// TwinCAT 3 PLC project Tests
// ProgramVersion: 3.1.4023.0
// libraries:
//   Tc2_Standard, * (Beckhoff Automation GmbH)
//   Tc2_System, * (Beckhoff Automation GmbH)
//   Tc3_Module, * (Beckhoff Automation GmbH)
// project tree:
//   DUTs/Alias/ T_Bool.TcDUT, T_Enum.TcDUT, T_SimpleStruct.TcDUT, T_PackedFb.TcDUT, T_String.TcDUT, T_Lreal.TcDUT, T_Dint.TcDUT, T_Wstring.TcDUT
//   DUTs/Enums/ E_Enum.TcDUT
//   DUTs/Struct/ ST_Simple.TcDUT, ST_Packed.TcDUT, ST_Complex.TcDUT, ST_STRUCT.TcDUT
//   DUTs/Unions/ U_Simple.TcDUT
//   / PlcTask.TcTTO
//   POUs/FBs/ FB_Invokable.TcPOU, FB_Simple.TcPOU, FB_Complex.TcPOU, FB_Packed.TcPOU
//   POUs/ P_Benchmark.TcPOU, P_Invoke.TcPOU, P_Notifications.TcPOU, P_Read.TcPOU, P_Write.TcPOU
// real-time tasks:
//   TASK PlcTask: cycle T#10ms, priority 8, ADS port 350
//   TASK FreeTask: cycle T#10ms, priority 6, ADS port 301

CONFIGURATION Tests
    RESOURCE PLC ON TwinCAT3
        TASK PlcTask(INTERVAL := T#10ms, PRIORITY := 8);
        PROGRAM P_Read WITH PlcTask : P_Read;
        PROGRAM P_Write WITH PlcTask : P_Write;
        PROGRAM P_Invoke WITH PlcTask : P_Invoke;
        PROGRAM P_Notifications WITH PlcTask : P_Notifications;
        PROGRAM P_Benchmark WITH PlcTask : P_Benchmark;
    END_RESOURCE
END_CONFIGURATION

// ---- DUTs/Alias/T_Bool.TcDUT
TYPE T_Bool : BOOL; END_TYPE

// ---- DUTs/Alias/T_Enum.TcDUT
TYPE T_Enum : E_Enum; END_TYPE

// ---- DUTs/Alias/T_SimpleStruct.TcDUT
TYPE T_SimpleStruct : ST_Simple; END_TYPE

// ---- DUTs/Alias/T_PackedFb.TcDUT
TYPE T_PackedFb : FB_Packed; END_TYPE

// ---- DUTs/Alias/T_String.TcDUT
TYPE T_String : STRING; END_TYPE

// ---- DUTs/Alias/T_Lreal.TcDUT
TYPE T_Lreal : LREAL; END_TYPE

// ---- DUTs/Alias/T_Dint.TcDUT
TYPE T_Dint : DINT; END_TYPE

// ---- DUTs/Alias/T_Wstring.TcDUT
TYPE T_Wstring : WSTRING; END_TYPE

// ---- DUTs/Enums/E_Enum.TcDUT
{attribute 'qualified_only'}
{attribute 'strict'}
TYPE E_Enum :
(
	Member0 := 0,
	Member1,
	Member2
);
END_TYPE

// ---- DUTs/Struct/ST_Simple.TcDUT
TYPE ST_Simple :
STRUCT
	bMember  		: BOOL;
    dtMember 		: DT;
	nMember   		: DINT;
END_STRUCT
END_TYPE

// ---- DUTs/Struct/ST_Packed.TcDUT
{attribute 'pack_mode' := '1'} 
TYPE ST_Packed :
STRUCT
	bMember  		: BOOL;
    dtMember 		: DT;
	fMember   		: LREAL;
END_STRUCT
END_TYPE

// ---- DUTs/Struct/ST_Complex.TcDUT
TYPE ST_Complex :
STRUCT
	bMember 		: BOOL;
	eMember 		: E_Enum;
	stSimpleMember 	: ST_Simple;
    stPackedMember 	: ST_Packed;
	fbMember 		: FB_Simple(TRUE, 99, 'Complex Test.');
	arrfMember 		: ARRAY[0..2] OF LREAL;
END_STRUCT
END_TYPE

// ---- DUTs/Struct/ST_STRUCT.TcDUT
TYPE ST_STRUCT :
STRUCT
	bVar  : BOOL;
	dtVar : DT;
	fVar  : LREAL;
END_STRUCT
END_TYPE

// ---- DUTs/Unions/U_Simple.TcDUT
TYPE U_Simple :
UNION
	bMember  		: BOOL;
    dtMember 		: DT;
	nMember   		: DINT;
END_UNION
END_TYPE

// ---- POUs/P_Read.TcPOU
PROGRAM P_Read
VAR
	bBoolean 		: BOOL 						:= TRUE;
	t_Bool 			: T_Bool 					:= TRUE;
	            	        					
	nByte 			: BYTE 						:= 32;
	nWord 			: WORD 						:= 31_234;
	nDword 			: DWORD 					:= 400_001;
	nLword 			: LWORD						:= 1_872_635_651_236;
	nSint 			: SINT 						:= -58;
	nUsint 			: USINT 					:= 254;
	nInt 			: INT						:= -32_688;
	nUint 			: UINT 						:= 65_456;
	nDint 			: DINT						:= -321_000_865;
	t_Dint 			: T_Dint 					:= -1_000_000_234;
	nUdint 			: UDINT						:= 4_268_999_001;
	nLint 			: LINT 						:= -18_000_100_020_003;
	nUlint 			: ULINT 					:= 45_000_100_020_003;
	
	nIntSubRange 	: INT(-4000..4000) 			:= -3996;
	
	fReal 			: REAL						:= -3.14;
	fLreal 			: LREAL						:= 44E2;
	t_Lreal 		: T_Lreal					:= 1.2E-2;
	
	sCleanString 	: STRING 					:= 'Hello World!';
	sDirtyString 	: STRING 					:= sCleanString;
	wsCleanString 	: WSTRING 					:= "Hello World!";
	wsDirtyString 	: WSTRING 					:= wsCleanString;
	t_String 		: T_String 					:= sCleanString;
	t_Wstring 		: T_Wstring 				:= wsCleanString;
	                                        	
	tTime 			: TIME 						:= T#4000MS;
	tLtime			: LTIME 					:= LTIME#12NS;
	dtDateTime 		: DT 						:= DT#2020-2-7-12:55:01;
	daDate 			: DATE 						:= DATE#2021-6-17;
	todTimeOfDay 	: TOD 						:= TOD#13:43:59.432;
	                                        	
	eEnum 			: E_Enum 					:= E_Enum.Member1;
	t_Enum 			: T_Enum					:= E_Enum.Member1;
	
	uSimple			: U_Simple					:= (nMember := 42);
	                                        	
	stSimple 		: ST_Simple 				:= (bMember := TRUE, dtMember := DT#2020-2-7-12:55:01, nMember := 448);
	stPacked 		: ST_Packed 				:= (bMember := TRUE, dtMember := DT#2023-3-10-15:30:01, fMember := 1.444);
	stComplex 		: ST_Complex 				:= (bMember := TRUE, eMember := E_Enum.Member2, stSimpleMember := stSimple, stPackedMember := stPacked, arrfMember := [1.23, 3.33, 1.11]);
	t_SimpleStruct 	: T_SimpleStruct			:= stSimple;
	
	fbSimple 		: FB_Simple(TRUE, -57, 'Simple Test.');
	fbPacked 		: FB_Packed 				:= (bMember := TRUE, nMember := 12, sMember := 'Packed Test.');
	fbComplex		: FB_Complex;
	t_PackedFb 		: T_PackedFb 				:= fbPacked;
	
	arrnInt 		: ARRAY[1..2] OF INT 		:= [-99, 99];
	arrfReal 		: ARRAY[1..3, 0..2] OF REAL := [2(10), 2(20), 2(30), 3(40)];
	ararfReal 		: ARRAY[0..2] OF ARRAY[0..2] OF REAL := [[3(10)], [3(20)], [3(30)]];
	arrarfReal 		: ARRAY[0..1, 0..2] OF ARRAY[0..2] OF LREAL := [3([3(11.5)]), 3([3(22.6)])];
	arrstComplex 	: ARRAY[0..1, 0..1] OF ST_Complex := [2(stComplex), 2(stComplex)];
	
	refBool 		: REFERENCE TO BOOL 		REF= bBoolean;
	refDint 		: REFERENCE TO DINT 		REF= nDint;
	refString 		: REFERENCE TO STRING 		REF= sCleanString;
	refWstring 		: REFERENCE TO WSTRING 		REF= wsCleanString;
	refTime 		: REFERENCE TO TIME 		REF= tTime;
	refDateTime 	: REFERENCE TO DT 			REF= dtDateTime;
	refDate 		: REFERENCE TO DATE 		REF= daDate;
	refTimeOfDay 	: REFERENCE TO TOD 			REF= todTimeOfDay;
	refEnum 		: REFERENCE TO E_Enum;
	refStruct 		: REFERENCE TO ST_Complex 	REF= stComplex;
	refFuncBlock 	: REFERENCE TO FB_Complex	REF= fbComplex;
	refArray 		: REFERENCE TO ARRAY[1..3, 0..2] OF REAL REF= arrfReal;
	refarrstComplex : REFERENCE TO ARRAY[0..1, 0..1] OF ST_Complex REF= arrstComplex;
	
	pBool 			: POINTER TO BOOL 			:= ADR(bBoolean);
	pDint 			: POINTER TO DINT 			:= ADR(nDint);
	pString 		: POINTER TO STRING 		:= ADR(sCleanString);
	pWstring 		: POINTER TO WSTRING 		:= ADR(wsCleanString);
	pTime 			: POINTER TO TIME 			:= ADR(tTime);
	pDateTime 		: POINTER TO DT 			:= ADR(dtDateTime);
	pDate 			: POINTER TO DATE 			:= ADR(daDate);
	pTimeOfDay 		: POINTER TO TOD 			:= ADR(todTimeOfDay);
	pEnum 			: POINTER TO E_Enum			:= ADR(eEnum);
	pStruct 		: POINTER TO ST_Complex 	:= ADR(stComplex);
	pFuncBlock 		: POINTER TO FB_Complex		:= ADR(fbComplex);
	pArray 			: POINTER TO ARRAY[1..3, 0..2] OF REAL := ADR(arrfReal);
	parrstComplex 	: POINTER TO ARRAY[0..1, 0..1] OF ST_Complex := ADR(arrstComplex);
END_VAR

sDirtyString := 'Ahh!';
wsDirtyString := "Ahh!";
refEnum REF= eEnum; // This is here because the compiler does not like initialising references to enums.

END_PROGRAM

// ---- POUs/FBs/FB_Simple.TcPOU
FUNCTION_BLOCK FB_Simple
VAR
	_bMember	: T_Bool := TRUE;
	_nMember 	: T_Dint := -57;
	_sMember 	: STRING := 'Testing Error.';
END_VAR

{attribute 'hide'}
METHOD FB_init : BOOL
VAR_INPUT
	bInitRetains : BOOL; // if TRUE, the retain variables are initialized (warm start / cold start)
	bInCopyCode : BOOL;  // if TRUE, the instance afterwards gets moved into the copy code (online change)
	bMember	: T_Bool;
	nMember : T_Dint;
	sMember : STRING;
END_VAR
THIS^._bMember := bMember;
THIS^._nMember := nMember;
THIS^._sMember := sMember;
END_METHOD

END_FUNCTION_BLOCK

// ---- POUs/FBs/FB_Packed.TcPOU
{attribute 'pack_mode' := '1'} 
FUNCTION_BLOCK FB_Packed
VAR_INPUT
	bMember	: T_Bool := TRUE;
	nMember : T_Dint := -57;
	sMember : STRING := 'Testing Error.';
END_VAR

END_FUNCTION_BLOCK

// ---- POUs/FBs/FB_Complex.TcPOU
FUNCTION_BLOCK FB_Complex
VAR
	_fMember 		: LREAL := 67.5;
	_stMember 		: ST_Complex := (bMember := TRUE, eMember := E_Enum.Member2, arrfMember := [1.23, 3.33, 1.11]); 
	_fbSimpleMember : FB_Simple(TRUE, 78, 'Complex Test.');
	_fbPackedMember : FB_Packed;
END_VAR

END_FUNCTION_BLOCK

// ---- POUs/P_Write.TcPOU
PROGRAM P_Write
VAR
	bBoolean 		: BOOL;
	t_Bool 			: T_Bool;
	refBool 		: REFERENCE TO BOOL 		REF= bBoolean;
	pBool 			: POINTER TO BOOL 			:= ADR(bBoolean);
	
	nDint 			: DINT;
	t_Dint 			: T_Dint;
	refDint 		: REFERENCE TO DINT 		REF= nDint;
	pDint 			: POINTER TO DINT 			:= ADR(t_Dint);
	
	fLreal 			: LREAL;
	t_Lreal 		: T_Lreal;
	refLreal 		: REFERENCE TO LREAL 		REF= fLreal;
	pLreal 			: POINTER TO LREAL 			:= ADR(t_Lreal);
	
	sString 		: STRING;
	t_String 		: T_String;
	refString 		: REFERENCE TO STRING 		REF= sString;
	pString 		: POINTER TO STRING 		:= ADR(t_String);
	
	wsString 		: WSTRING;
	t_Wstring 		: T_WString;
	refWstring 		: REFERENCE TO WSTRING 		REF= wsString;
	pWstring 		: POINTER TO WSTRING 		:= ADR(t_Wstring);
	
	tTime 			: TIME;
	refTime 		: REFERENCE TO TIME 		REF= tTime;
	pTime 			: POINTER TO TIME 			:= ADR(tTime);
	
	tLtime			: LTIME;
	refLtime		: REFERENCE TO LTIME 		REF= tLtime;
	pLTime			: POINTER TO LTIME 			:= ADR(tLtime);
	
	dtDateTime 		: DT;
	refDateTime 	: REFERENCE TO DT 			REF= dtDateTime;
	pDateTime 		: POINTER TO DT 			:= ADR(dtDateTime);
	
	daDate 			: DATE;
	refDate 		: REFERENCE TO DATE 		REF= daDate;
	pDate 			: POINTER TO DATE 			:= ADR(daDate);
	
	todTimeOfDay 	: TOD;
	refTimeOfDay 	: REFERENCE TO TOD 			REF= todTimeOfDay;
	pTimeOfDay 		: POINTER TO TOD 			:= ADR(todTimeOfDay);
	
	eEnum 			: E_Enum;
	t_Enum 			: T_Enum;
	refEnum 		: REFERENCE TO E_Enum;
	pEnum 			: POINTER TO E_Enum			:= ADR(t_Enum);
	
	stSimple 		: ST_Simple;
	stPacked 		: ST_Packed;
	stComplex 		: ST_Complex;
	t_Struct 		: T_SimpleStruct;
	refStruct		: REFERENCE TO ST_Complex 	REF= stComplex;
	pStruct 		: POINTER TO ST_Complex 	:= ADR(stComplex);
	
	fbSimple 		: FB_Simple(0, 0, '');
	fbPacked 		: FB_Packed;
	fbComplex		: FB_Complex;
	t_PackedFb 		: T_PackedFb;
	refFuncBlock 	: REFERENCE TO FB_Complex	REF= fbComplex;
	pFuncBlock 		: POINTER TO FB_Complex		:= ADR(fbComplex);
	
	arrnInt 		: ARRAY[1..2] OF INT;
	arrfReal 		: ARRAY[1..3, 0..2] OF REAL;
	ararfReal 		: ARRAY[0..2] OF ARRAY[0..2] OF REAL;
	arrarfReal 		: ARRAY[0..1, 0..2] OF ARRAY[0..2] OF LREAL;
	arrstComplex 	: ARRAY[0..1, 0..1] OF ST_Complex;
	arfbSimple		: ARRAY[0..2] OF FB_Simple[(FALSE, 0, '')];
	refArray 		: REFERENCE TO ARRAY[1..3, 0..2] OF REAL REF= arrfReal;
	refarrstComplex : REFERENCE TO ARRAY[0..1, 0..1] OF ST_Complex REF= arrstComplex;
	pArray 			: POINTER TO ARRAY[1..3, 0..2] OF REAL := ADR(arrfReal);
	parrstComplex 	: POINTER TO ARRAY[0..1, 0..1] OF ST_Complex := ADR(arrstComplex);
END_VAR

refEnum REF= eEnum; // This is here because the compiler does not like initialising references to enums.

END_PROGRAM

// ---- POUs/P_Invoke.TcPOU
PROGRAM P_Invoke
VAR
	fbInvoke : FB_Invokable;
END_VAR

{attribute 'TcRpcEnable'}
METHOD Meth : INT
VAR_INPUT
	Value : INT;
END_VAR
Meth := Value*2;
END_METHOD

END_PROGRAM

// ---- POUs/FBs/FB_Invokable.TcPOU
FUNCTION_BLOCK FB_Invokable
VAR
END_VAR

{attribute 'TcRpcEnable'}
METHOD Test : INT
VAR_IN_OUT
	Value :  INT;
	Value2 : INT;
END_VAR
Test 	:= Value * 2;
Value 	:= Test * 2;
Value2 	:= Value * 2;
END_METHOD

END_FUNCTION_BLOCK

// ---- POUs/P_Notifications.TcPOU
PROGRAM P_Notifications
VAR
END_VAR

END_PROGRAM

// ---- POUs/P_Benchmark.TcPOU
PROGRAM P_Benchmark
VAR
	stValue 		: ST_Simple;
	stComplexValue	: ST_Complex;
	fbValue			: FB_Simple(TRUE, 12, 'Simple function block.');
	fbComplexValue 	: FB_Complex;
	ardtValues		: ARRAY[0..999] OF DT			:= [1000(DT#2024-12-7-11:45:56)];
	arfValues		: ARRAY[0..999] OF LREAL		:= [1000(3.14)];
	arsValues		: ARRAY[0..999] OF WSTRING		:= [1000("Hello there!")];
	arstStruct		: ARRAY[0..999] OF ST_STRUCT	:= [1000((bVar := TRUE, dtVar := DT#2020-2-7-12:55:01, fVar := 3.14))];
	arstValues		: ARRAY[0..999] OF ST_Simple 	:= [2((bMember := TRUE, dtMember := DT#2020-2-7-12:55:01, nMember := 448))];
	arfbValues 		: ARRAY[0..999] OF FB_Simple[(TRUE, -87, 'Test simple array.')];
END_VAR

END_PROGRAM
